// TIA Portal V17 export
// export: Created 2025-03-05T08:02:28.5308012Z, ExportSetting WithDefaults, DisplayName Totally Integrated Automation Portal, DisplayVersion V17 Update 8, DisplayName TIA Portal Openness, DisplayVersion V17 Update 8, DisplayName TIA Portal Version Control Interface, DisplayVersion V17, DisplayName SINAMICS Startdrive Advanced, DisplayVersion V17 SP2, DisplayName SINAMICS Startdrive G110M, G120, G120C, G120D, G120P, G115D, DisplayVersion V17 SP2, DisplayName SINAMICS Startdrive G130, G150, S120, S150, SINAMICS MV, S210, DisplayVersion V17 SP2, DisplayName STEP 7 Professional, DisplayVersion V17 Update 8, DisplayName SINUMERIK ONE STEP 7 Toolbox, DisplayVersion V17 Update 12, DisplayName SINUMERIK 840D sl STEP 7 Toolbox, DisplayVersion V17 Update 12, DisplayName STEP 7 Safety, DisplayVersion V17 Update 6, DisplayName WinCC Advanced, DisplayVersion V17 Update 8
TYPE "PYROMETER"
// stored: IsFailsafeCompliant false
   STRUCT
      PYROMETER_READY_INPUT : Bool;   // Pyrometer Ready Input
      PYROMETER_FAULT_INPUT : Bool;   // Pyrometer Fault Input
      START_GENERAL_CONDITIONS : Bool;   // Start General Conditions
      START_INITIAL_CONDITIONS : Bool;   // Start Initial Conditions
      START_MANUAL_REQUEST : Bool;   // Start Manual Request
      START_AUTO_REQUEST : Bool;   // Start Auto Request
      START_GLOBAL_REQUEST : Bool;   // Start Global Request
      START_COMMAND : Bool;   // Start Command
      STARTED : Bool;   // Started
      FEEDBACK_STARTED : Bool;   // Feedback Started
      STOP_GENERAL_CONDITIONS : Bool;   // Stop General Conditions
      STOP_INITIAL_CONDITIONS : Bool;   // Stop Initial Conditions
      STOP_MANUAL_REQUEST : Bool;   // Stop Manual Request
      STOP_AUTO_REQUEST : Bool;   // Stop Auto Request
      STOP_GLOBAL_REQUEST : Bool;   // Stop Global Request
      STOP_COMMAND : Bool;   // Stop Command
      STOPPED : Bool;   // Stopped
      FEEDBACK_STOP : Bool;   // Feedback Stop
      SPARE_BYTE_4 : Byte;   // Spare Byte 4
      DIFERENCIAL_PROTECTION_FAULT : Bool;   // Diferential Protection Fault
      CIRCUIT_BRAKER_FAULT : Bool;   // Circuit Breaker Fault
      CONTACTOR_FEEDBACK_FAULT : Bool;   // Contactor Feedback Fault
      SAFETY_FEEDBACK_FAULT : Bool;   // Safety Feedback Fault
      FEEDBACK_FAULT : Bool;   // Feedback Fault
      ERROR_FAULT : Bool;   // Error Fault
      NOT_RUNNING_ALARM : Bool;   // Not Running Alarm
      PRESSURE_1 : Bool;   // Pressure_1
      AUX0 : Bool;   // Aux0
      AUX1 : Bool;   // Aux1
      AUX2 : Bool;   // Aux2
      AUX3 : Bool;   // Aux3
      WARNING_GONE : Bool;   // Warning Gone
      AUX5 : Bool;   // Aux5
      AUX6 : Bool;   // Aux6
      AUX7 : Bool;   // Aux7
      START_GENERAL_CONDITIONS_HELP : Bool;   // Start General Conditions Help
      START_INITIAL_CONDITIONS_HELP : Bool;   // Start Initial Conditions Help
      STOP_GENERAL_CONDITIONS_HELP : Bool;   // Stop General Conditions Help
      STOP_INITIAL_CONDITIONS_HELP : Bool;   // Stop Initial Conditions Help
      FAULT : Bool;   // Fault
   END_STRUCT;
END_TYPE
